{attribute 'qualified_only'}
VAR_GLOBAL
	aMeterData: ARRAY[1..20] OF ST_PowerMeter;
END_VAR

(* stored: Version 1.1.0.1, ProductVersion 3.1.4024.12
   GVL GVL: Id {f60b7de8-9674-45d0-b6f3-b6573daddec5} *)
